{attribute 'GeneratedUsingTerminal: KL9900-0056'}
{attribute addProperty BoxType "KL9900-0056"}
{attribute addProperty Description ""}
{attribute addProperty Physics ""}
{attribute addProperty Id "Channel_1AT %Q*Channel_2E0D480D0"}
{attribute addProperty CRC "104794512"}
{attribute addProperty Size "0"}
TYPE KL_063F0990 :
STRUCT
	{attribute addProperty Name "Channel_1"}
	Channel_1 : Channel_2E0D480D;
END_STRUCT
END_TYPE

(* stored: Version 1.2.0.0, ProductVersion 3.1.4024.11
   DUT KL_063F0990: Id {691249e3-9de5-47f9-aad1-4c51212f3a2c} *)
